ABB RobotStudio station: Session1.rspag

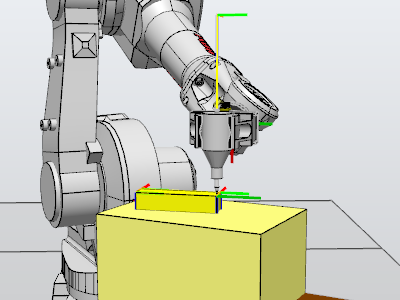
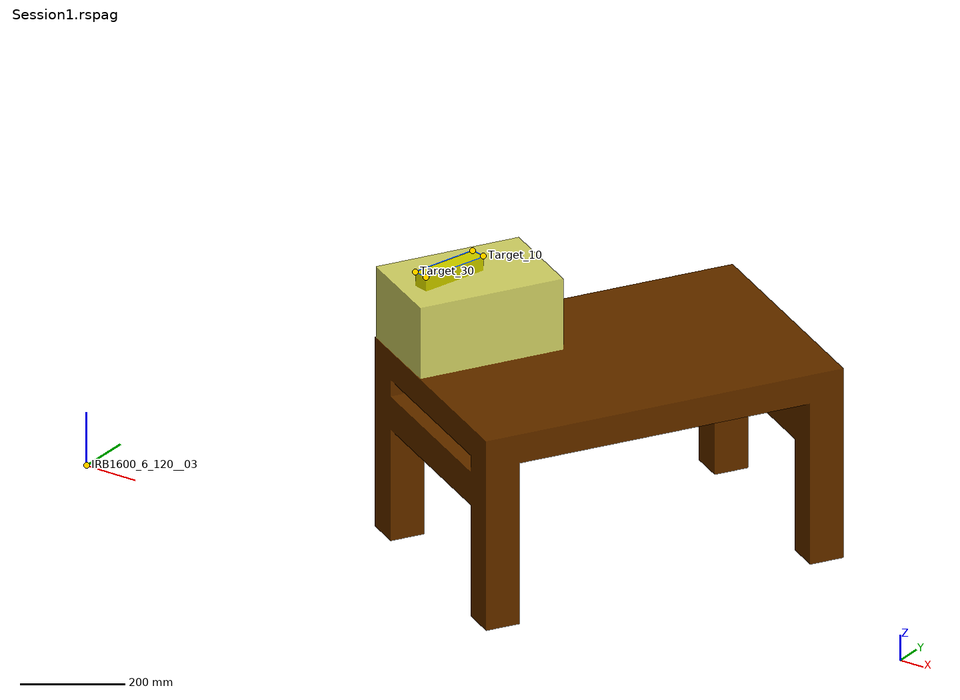
[picture v1: parts stored in the station drawn from their meshes, with robot base, taught points and paths (robot models come from the ABB library and are not in the file)]
--- station ---
Station Session1 (saved by RobotStudio 24.2.10821.1)
Controller Controller1
  mechanical unit ROB_1: IRB1600_6_120__03, 6 joints, base frame (0, 0, 0) mm
Layout (positions relative to the parent item):
  - IRB1600_6_120__03 [mechanism, from %ABB.RobotStudio.Models.IRB1600%\IRB1600_6_120_G_03.rslib] at (0, 0, 0) mm; joint values [0.4143, -0.1069, 0.5714, -2.0801, 0.799, 2.246] (rad or m)
  - Pen [mechanism, from Training Objects\Pen.rslib] at (644.76, 239.07, 690) mm, rotated rx 0 ry 90 rz -15 deg
  - IRC5_Control-Module [part, from %ABB.RobotStudio.Models.IRC5%\IRC5_Control-Module.rslib] at (-1161.73, -1082.62, 100) mm, rotated rx 90 ry 0 rz 90 deg
  - Table [part] at (600, 100, 0) mm, rotated rx 0 ry 0 rz -30 deg, size 500 x 750 x 400 mm
  - Box [part] at (601.78, 100.13, 400) mm, rotated rx 0 ry 0 rz -29.85 deg, size 200 x 300 x 180 mm
Attachment: Pen is attached to IRB1600_6_120__03 / Link6
Targets, tools, work objects and paths stored in the station and not in the controller backup, written as RAPID:
! task T_ROB1
MODULE Module1
  CONST robtarget pBox_10:=[[779.99,202.836,580],[0,0.130526192,0.991444861,0],[0,-2,1,0],[9E+09,9E+09,9E+09,9E+09,9E+09,9E+09]];
  CONST robtarget pBox_20:=[[749.085,211.136,580],[0,0.130526192,0.991444861,0],[0,-2,1,0],[9E+09,9E+09,9E+09,9E+09,9E+09,9E+09]];
  CONST robtarget pBox_30:=[[712.252,73.996,580],[0,0.130526192,0.991444861,0],[0,-2,1,0],[9E+09,9E+09,9E+09,9E+09,9E+09,9E+09]];
  CONST robtarget pBox_40:=[[743.157,65.696,580],[0,0.130526192,0.991444861,0],[0,-2,1,0],[9E+09,9E+09,9E+09,9E+09,9E+09,9E+09]];
  CONST robtarget Appr_Box:=[[779.99,202.836,880],[0,0.130526192,0.991444861,0],[0,-1,0,0],[9E+09,9E+09,9E+09,9E+09,9E+09,9E+09]];
ENDMODULE


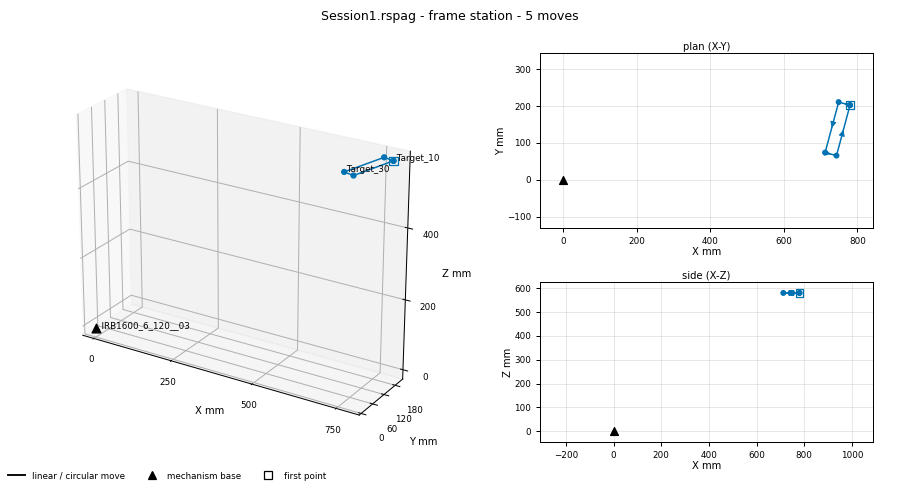
[picture p0: tool path of Session1.rspag in frame station, 5 of 5 moves have a stored position in this frame; points joined in program order, loops and branches not executed]
--- Backups/Controller1/RAPID/TASK1/PROGMOD/CalibData.mod ---
MODULE CalibData
    PERS tooldata Pen_TCP:=[TRUE,[[110,0,140],[0.707106781,0,0.707106781,0]],[1,[10.7435139,0,140],[1,0,0,0],0,0,0]];
    TASK PERS wobjdata Wobj_Box:=[FALSE,TRUE,"",[[0,0,0],[1,0,0,0]],[[0,0,0],[1,0,0,0]]];
ENDMODULE

--- Backups/Controller1/RAPID/TASK1/PROGMOD/Module1.mod ---
MODULE Module1
        CONST robtarget Target_10:=[[779.99,202.836,580],[0,0.130526192,0.991444861,0],[0,-2,1,0],[9E+09,9E+09,9E+09,9E+09,9E+09,9E+09]];
    CONST robtarget Target_20:=[[749.085,211.136,580],[0,0.130526192,0.991444861,0],[0,-2,1,0],[9E+09,9E+09,9E+09,9E+09,9E+09,9E+09]];
    CONST robtarget Target_30:=[[712.252,73.996,580],[0,0.130526192,0.991444861,0],[0,-2,1,0],[9E+09,9E+09,9E+09,9E+09,9E+09,9E+09]];
    CONST robtarget Target_40:=[[743.157,65.696,580],[0,0.130526192,0.991444861,0],[0,-2,1,0],[9E+09,9E+09,9E+09,9E+09,9E+09,9E+09]];
!***********************************************************
    !
    ! Module:  Module1
    !
    ! Description:
    !   <Insert description here>
    !
    ! Author: ahmadk
    !
    ! Version: 1.0
    !
    !***********************************************************


    !***********************************************************
    !
    ! Procedure main
    !
    !   This is the entry point of your program
    !
    !***********************************************************
    PROC main()
        !Add your code here
        Path_Box;
    ENDPROC
    PROC Path_Box()
        MoveL Target_10,v300,fine,Pen_TCP\WObj:=Wobj_Box;
        MoveL Target_20,v300,fine,Pen_TCP\WObj:=Wobj_Box;
        MoveL Target_30,v300,fine,Pen_TCP\WObj:=Wobj_Box;
        MoveL Target_40,v300,fine,Pen_TCP\WObj:=Wobj_Box;
        MoveL Target_10,v300,fine,Pen_TCP\WObj:=Wobj_Box;
    ENDPROC
ENDMODULE
